(* PLC project mixing, Dassault Systèmes ControlBuild 2024x *)
(* stored: creationDateTime 2023-10-03T11:13:42-01:00 *)

PROGRAM bottling_line.mixing
  VAR_INPUT
    autoMode : BOOL := false;
    manualMode : BOOL := false;
  END_VAR
  VAR_INPUT
    acknowledgePB : BOOL := false;
  END_VAR
  VAR_INPUT
    fillingValve : BOOL := false;
    hiSpeedAgitator : BOOL := false;
    loSpeedAgitator : BOOL := false;
  END_VAR
  VAR_INPUT
    inputFlow : REAL := 0.0;
  END_VAR
  VAR_OUTPUT
    highLevel : BOOL := false;
    lowLevel : BOOL := false;
  END_VAR
  VAR_OUTPUT
    level : REAL := 0.0;
    outputFlow : REAL := 0.0;
  END_VAR

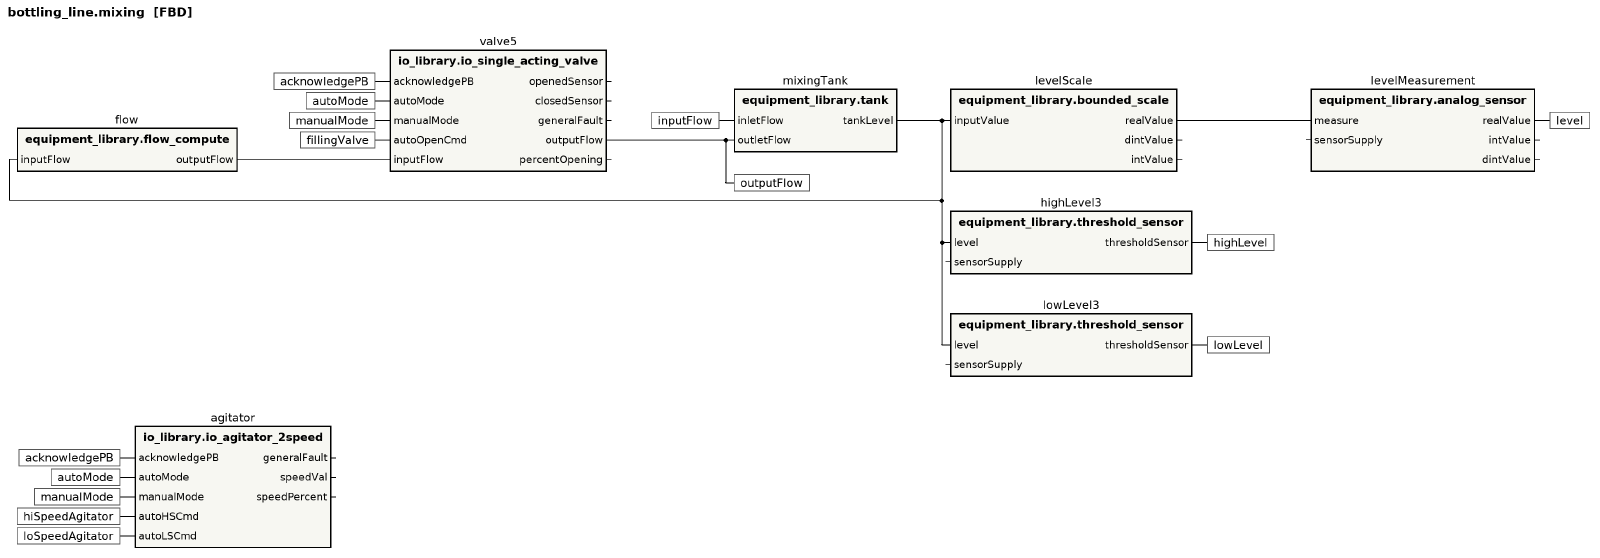
(* FBD diagram, written out as Structured Text *)
flow(inputFlow := mixingTank.tankLevel);
valve5(acknowledgePB := acknowledgePB, autoMode := autoMode, manualMode := manualMode, autoOpenCmd := fillingValve, inputFlow := flow.outputFlow);
mixingTank(inletFlow := inputFlow, outletFlow := valve5.outputFlow);
levelScale(inputValue := mixingTank.tankLevel);
levelMeasurement(measure := levelScale.realValue);
level := levelMeasurement.realValue;
highLevel3(level := mixingTank.tankLevel);
highLevel := highLevel3.thresholdSensor;
lowLevel3(level := mixingTank.tankLevel);
lowLevel := lowLevel3.thresholdSensor;
outputFlow := valve5.outputFlow;
agitator(acknowledgePB := acknowledgePB, autoMode := autoMode, manualMode := manualMode, autoHSCmd := hiSpeedAgitator, autoLSCmd := loSpeedAgitator);
END_PROGRAM
